SYSTEM TEST_TEXT (* Test of JTextPane-based components *)
  (* Standard: 61499-1 *)
  (* Version 0.1, 2007-03-31, JHC, Holobloc Inc, Corrected naming of resources and initial values. *)
  (* Version 0.0, 2004-06-20, JHC, Rockwell Automation *)
  APPLICATION APP1
  END_APPLICATION
  DEVICE DEV1 : FRAME_DEVICE(BOUNDS := [100,100,350,350], GRID := [2,1])
    RESOURCE STRINGS : PANEL_RESOURCE
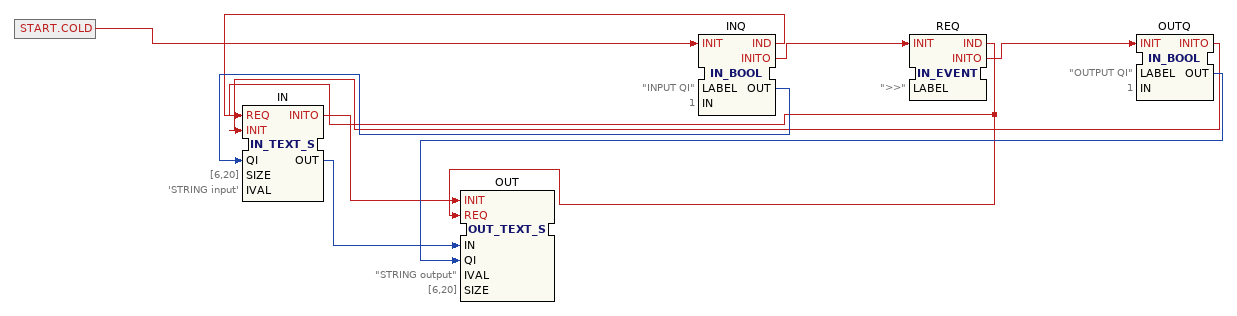
      FBS
        IN : IN_TEXT_S(SIZE := [6,20], IVAL := 'STRING input');
        OUT : OUT_TEXT_S(IVAL := "STRING output", SIZE := [6,20]);
        REQ : IN_EVENT(LABEL := ">>");
        INQ : IN_BOOL(LABEL := "INPUT QI", IN := 1);
        OUTQ : IN_BOOL(LABEL := "OUTPUT QI", IN := 1);
      END_FBS
      EVENT_CONNECTIONS
        REQ.IND TO IN.REQ;
        IN.INITO TO OUT.INIT;
        INQ.IND TO IN.REQ;
        REQ.IND TO OUT.REQ;
        INQ.INITO TO REQ.INIT;
        REQ.INITO TO OUTQ.INIT;
        START.COLD TO INQ.INIT;
        OUTQ.INITO TO IN.INIT;
      END_CONNECTIONS
      DATA_CONNECTIONS
        INQ.OUT TO IN.QI;
        IN.OUT TO OUT.IN;
        OUTQ.OUT TO OUT.QI;
      END_CONNECTIONS
    END_RESOURCE
    RESOURCE WSTRINGS : PANEL_RESOURCE
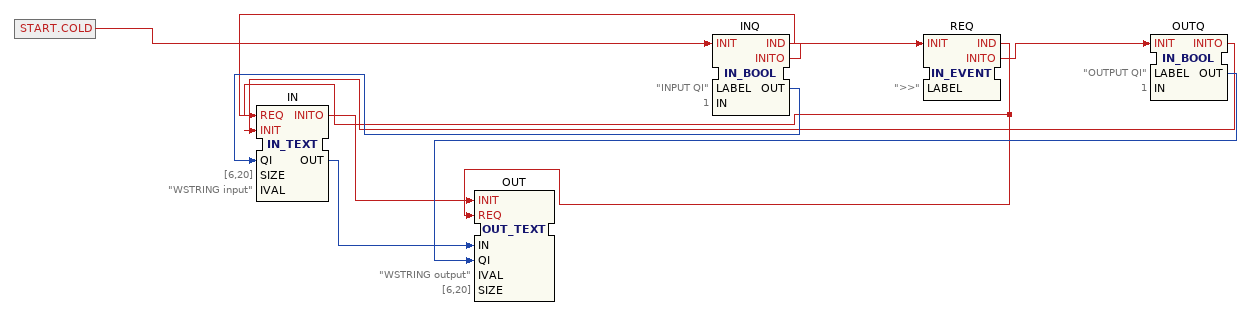
      FBS
        IN : IN_TEXT(SIZE := [6,20], IVAL := "WSTRING input");
        OUT : OUT_TEXT(IVAL := "WSTRING output", SIZE := [6,20]);
        REQ : IN_EVENT(LABEL := ">>");
        INQ : IN_BOOL(LABEL := "INPUT QI", IN := 1);
        OUTQ : IN_BOOL(LABEL := "OUTPUT QI", IN := 1);
      END_FBS
      EVENT_CONNECTIONS
        REQ.IND TO IN.REQ;
        IN.INITO TO OUT.INIT;
        INQ.IND TO IN.REQ;
        REQ.IND TO OUT.REQ;
        INQ.INITO TO REQ.INIT;
        REQ.INITO TO OUTQ.INIT;
        START.COLD TO INQ.INIT;
        OUTQ.INITO TO IN.INIT;
      END_CONNECTIONS
      DATA_CONNECTIONS
        INQ.OUT TO IN.QI;
        IN.OUT TO OUT.IN;
        OUTQ.OUT TO OUT.QI;
      END_CONNECTIONS
    END_RESOURCE
  END_DEVICE
END_SYSTEM
